// TwinCAT 3 PLC project OOP_PLC
// ProgramVersion: 3.1.4020.10
// libraries:
//   Tc2_Standard, * (Beckhoff Automation GmbH)
//   Tc2_System, * (Beckhoff Automation GmbH)
//   Tc3_Module, * (Beckhoff Automation GmbH)
//   VisuDialogs, * (System)
//   Tc3_System_DK,3.3.1.8,Beckhoff - DK
// project tree:
//   000 - General/ FB_RcvData.TcPOU, FB_RcvDataBuffer.TcPOU, GVL_MachineSettings.TcGVL, MAIN.TcPOU, P_System.TcPOU, visMain.TcVIS
//   010 - Machine Part 01/ FB_MachinePart01.TcPOU, ST_SettingMachinePart01.TcDUT, visSettingMachPart1.TcVIS
//   020 - Machine Part 02/ FB_MachinePart02.TcPOU, ST_SettingMachinePart02.TcDUT, visSettingMachPart2.TcVIS
//   100 - Network/ FB_CustomTcp.TcPOU, I_TcpClient.TcIO, I_TcpRcv.TcIO, SampleTcpClient.TcPOU, FB_SimpleTcpClient.TcPOU, SampleTcpServer.TcPOU, SampleUdpEchoServer.TcPOU, ST_Log.TcDUT, T_TcpRcv.TcDUT, U_IPAddr.TcDUT, U_Data.TcDUT
//   990 - NTO Standard/HResult/ F_Busy.TcPOU, F_Code.TcPOU, F_Fail.TcPOU, F_Success.TcPOU, GVL_HResultError.TcGVL, GVL_HResultSuccess.TcGVL
//   990 - NTO Standard/Object/ FB_Object.TcPOU, GVL_ObjectSetup.TcGVL, I_Object.TcIO, T_ErrorHistory.TcDUT
//   991 - NTO Actuators/010 - Cylinders/CylinderCollection/ FB_CylinderOneValveSpringRetX_2.TcPOU, FB_CylinderTwoValveRetX_3.TcPOU, txtCylinderTypes.TcTLO
//   991 - NTO Actuators/010 - Cylinders/ E_CylinderEnableMode.TcDUT, I_StandardCylinder.TcIO, ST_StandardCylinderSettings.TcDUT, txtLstCylinderEnableMode.TcTLO, visStandardCylinderSettings.TcVIS
//   991 - NTO Actuators/020 - Motors/MotorCollection/ FB_Motor.TcPOU, FB_MotorInverterFITYPE.TcPOU, txtMotorTypes.TcTLO
//   991 - NTO Actuators/020 - Motors/ E_MotorEnableMode.TcDUT, I_StandardMotor.TcIO, ST_StandardMotorSettings.TcDUT, txtLstMotorEnableMode.TcTLO, visStandardMotorSettings.TcVIS
//   / GlobalTextList.TcGTLO, PlcTask.TcTTO, Visualization Manager.TcVMO (not stored)
// real-time tasks:
//   TASK PlcTask: cycle T#1ms, priority 20, ADS port 350
//   TASK VISU_TASK: cycle T#200000us, priority 30, ADS port 351
// I/O:
//   DEVICE Device 1 (RT-Ethernet Adapter)

CONFIGURATION OOP_PLC
    RESOURCE PLC ON TwinCAT3
        TASK PlcTask(INTERVAL := T#1ms, PRIORITY := 20);
        PROGRAM MAIN WITH PlcTask : MAIN;
    END_RESOURCE
END_CONFIGURATION

// ---- 010 - Machine Part 01/ST_SettingMachinePart01.TcDUT
TYPE ST_SettingMachinePart01 :
STRUCT
    nMotorType : BYTE; //Motor type
    stMotorSettings : ST_StandardMotorSettings;
    nCylinderType : BYTE; //Cylinder type
    stCylinderSettings : ST_StandardCylinderSettings;
END_STRUCT
END_TYPE

// ---- 020 - Machine Part 02/ST_SettingMachinePart02.TcDUT
TYPE ST_SettingMachinePart02 :
STRUCT
    nCylinder1Type : BYTE; //Cylinder type
    stCylinder1Settings : ST_StandardCylinderSettings;
    nCylinder2Type : BYTE; //Cylinder type
    stCylinder2Settings : ST_StandardCylinderSettings;
END_STRUCT
END_TYPE

// ---- 100 - Network/ST_Log.TcDUT
TYPE ST_Log :
STRUCT
	nSocketID : UDINT;
	eTcpEvent : TCPIP_EVENT;
	sMessage : STRING;
END_STRUCT
END_TYPE

// ---- 100 - Network/T_TcpRcv.TcDUT
TYPE T_TcpRcv : POINTER TO FB_RcvDataBuffer; END_TYPE

// ---- 100 - Network/U_IPAddr.TcDUT
TYPE U_IPAddr :
UNION
	aIpAddr : ARRAY[0..3] OF BYTE;
	nIpAddr : UDINT;
END_UNION
END_TYPE

// ---- 100 - Network/U_Data.TcDUT
TYPE U_Data :
UNION
	sData : STRING(255);
	aData : ARRAY[0..255] OF BYTE;
END_UNION
END_TYPE

// ---- 990 - NTO Standard/Object/T_ErrorHistory.TcDUT
///Error history type
TYPE T_ErrorHistory : ARRAY[GVL_ObjectSetup.cErrorHistMin..GVL_ObjectSetup.cErrorHistMax] OF DWORD; END_TYPE

// ---- 991 - NTO Actuators/010 - Cylinders/E_CylinderEnableMode.TcDUT
{attribute 'qualified_only'}
{attribute 'strict'}
///Cylinder enable mode
TYPE E_CylinderEnableMode :
(
    eCylEnaOff,         ///Enable does not affect cylinder
	eCylEnaToHome,      ///When enable false, move cylinder to home
    eCylEnaToOut,       ///When enable false, move cylinder to out
    eCylEnaNoChanges    ///When enable false, cylinder keeps the position
);
END_TYPE

// ---- 991 - NTO Actuators/010 - Cylinders/ST_StandardCylinderSettings.TcDUT
///Standard cylinder settings
TYPE ST_StandardCylinderSettings :
STRUCT
    bSensorAtOut : BOOL; ///Cylinder has sensor at out
    tTimeToOrAtOut : TIME; ///Cylinder at or to out, bSensorOut = true: at out, bSensorOut = false: to out 
    bSensorAtHome : BOOL; ///Cylinder has sensor at home
    tTimeToOrAtHome : TIME; ///Cylinder at or to home, bSensorOut = true: at home, bSensorOut = false: to home
    eEnableMode : E_CylinderEnableMode; ///Cylinder enable mode
END_STRUCT
END_TYPE

// ---- 991 - NTO Actuators/020 - Motors/E_MotorEnableMode.TcDUT
{attribute 'qualified_only'}
{attribute 'strict'}
///Cylinder enable mode
TYPE E_MotorEnableMode :
(
    eMotorEnaOff,       ///Enable does not affect motor
    eMotorEnaAll,       ///When enable false, motor cannot move CW or CCW
    eMotorEnaAllowCW,   ///When enable false, motor can onlu move CW
    eMotorEnaAllowCCW   ///When enable false, motor can onlu move CCW   
);
END_TYPE

// ---- 991 - NTO Actuators/020 - Motors/ST_StandardMotorSettings.TcDUT
///Standard motor settings
TYPE ST_StandardMotorSettings :
STRUCT
    eEnableMode : E_MotorEnableMode; ///Enable mode
    nMaxSpeed : UINT; //Max speed in 0.1%
    nMaxAcc : UINT; //Max accelaration in FI dependent type
    nMaxDec : UINT; //Max deceleration in FI dependent type
END_STRUCT
END_TYPE

// ---- 000 - General/GVL_MachineSettings.TcGVL
{attribute 'qualified_only'}
VAR_GLOBAL PERSISTENT
    stSettingsMach01_1 : ST_SettingMachinePart01 := (nMotorType := 0, nCylinderType := 1);
    stSettingsMach01_2 : ST_SettingMachinePart01 := (nMotorType := 1, nCylinderType := 0);
    stSettingsMach02_1 : ST_SettingMachinePart02 := (
		nCylinder1Type := 0, stCylinder1Settings := (bSensorAtOut := TRUE, eEnableMode := E_CylinderEnableMode.eCylEnaToHome),
		nCylinder2Type := 1, stCylinder2Settings := (bSensorAtOut := FALSE, eEnableMode := E_CylinderEnableMode.eCylEnaToOut));
    stSettingsMach02_2 : ST_SettingMachinePart02 := (nCylinder1Type := 1, nCylinder2Type := 0);
END_VAR

// ---- 990 - NTO Standard/HResult/GVL_HResultError.TcGVL
{attribute 'qualified_only'}
VAR_GLOBAL CONSTANT
    cHR_ErrGeneral : HRESULT := UDINT_TO_DINT(16#A0000000); //Fail with general error
    cHR_ErrInvalidParameter : HRESULT := UDINT_TO_DINT(16#A0000001); //Fail with invalid parameters    
	cHR_ErrConnect : HRESULT := UDINT_TO_DINT(16#A0000002); //Fail, when trying to connect
	cHR_ErrAllocSocket : HRESULT := UDINT_TO_DINT(16#A0000003); //Fail, when allocating a socket
	cHR_ErrNotConnected : HRESULT := UDINT_TO_DINT(16#A0000002); //Fail, not connected
END_VAR

// ---- 990 - NTO Standard/HResult/GVL_HResultSuccess.TcGVL
{attribute 'qualified_only'}
VAR_GLOBAL CONSTANT
    cHR_SuccesDone : HRESULT := 16#20000001; //Successfully done
    cHR_SuccesBusy : HRESULT := 16#20000002; //Busy, keep calling to wait for done or error    
END_VAR

// ---- 990 - NTO Standard/Object/GVL_ObjectSetup.TcGVL
{attribute 'qualified_only'}
VAR_GLOBAL CONSTANT
    cErrorHistMin : INT := 0; ///Error history array bound minimum
    cErrorHistMax : INT := 10; ///Error history array bound maximum
END_VAR

// ---- 100 - Network/I_TcpClient.TcIO
{attribute 'c++_compatible'}
INTERFACE I_TcpClient EXTENDS I_Object

METHOD PUBLIC Connect : HRESULT
VAR_INPUT
	uIPAddr : U_IPAddr;
	nPort : UINT;
	{warning 'Implemented with POINTER TO, until Beckhoff comes with solution to why Interface call crashes app'}
	ipRcvData : T_TcpRcv;//I_TcpRcv; 
END_VAR
END_METHOD

PROPERTY DataLogging : BOOL
GET
END_GET
SET
END_SET
END_PROPERTY

METHOD PUBLIC Disconnect : HRESULT
VAR_INPUT
END_VAR
END_METHOD

PROPERTY EventLogging : BOOL
GET
END_GET
SET
END_SET
END_PROPERTY

PROPERTY IpAddress : U_IPAddr
GET
END_GET
END_PROPERTY

PROPERTY IsConnected : BOOL
GET
END_GET
END_PROPERTY

PROPERTY Port : UINT
GET
END_GET
END_PROPERTY

METHOD SendData : HRESULT
VAR_INPUT
	nData : UDINT;
	pData : PVOID;
END_VAR
END_METHOD

PROPERTY SendingData : BOOL
GET
END_GET
END_PROPERTY

END_INTERFACE

// ---- 100 - Network/I_TcpRcv.TcIO
{attribute 'c++_compatible'}
INTERFACE I_TcpRcv

METHOD NewData : HRESULT
VAR_INPUT
	nData	: UDINT;
	pData	: PVOID;
END_VAR
END_METHOD

END_INTERFACE

// ---- 990 - NTO Standard/Object/I_Object.TcIO
{attribute 'c++_compatible'}
///Base object interface
INTERFACE I_Object

//Cycle Task, do not override this methode cyclic code is placed in M_Control
METHOD CycleTask
VAR_INPUT
END_VAR
END_METHOD

///Error, do not implement property override
PROPERTY Error : BOOL
GET
END_GET
END_PROPERTY

///Error id, do not implement property override
PROPERTY ErrorID : DWORD
GET
END_GET
END_PROPERTY

///Pointer to error history, do not implement property override
PROPERTY Errors : POINTER TO T_ErrorHistory
GET
END_GET
END_PROPERTY

///Name, do not implement property override
PROPERTY PUBLIC Name : String(50)
GET
END_GET
END_PROPERTY

///Reset error, allways call super
METHOD Reset
VAR_INPUT
END_VAR
END_METHOD

///Version,do not implement property override
PROPERTY PUBLIC Version : String(8)
GET
END_GET
END_PROPERTY

END_INTERFACE

// ---- 991 - NTO Actuators/010 - Cylinders/I_StandardCylinder.TcIO
{attribute 'c++_compatible'}
///Standard cylinder
INTERFACE I_StandardCylinder EXTENDS I_Object

///Cylinder at home position
PROPERTY AtHome : BOOL
GET
END_GET
END_PROPERTY

///Cylinder at out position
PROPERTY AtOut : BOOL
GET
END_GET
END_PROPERTY

///Enable cylinder to change position
PROPERTY Enable : BOOL
GET
END_GET
SET
END_SET
END_PROPERTY

METHOD MoveHome
VAR_INPUT
END_VAR
END_METHOD

METHOD MoveOut
VAR_INPUT
END_VAR
END_METHOD

///Pointer to settings, should be set at FB_init but can be modified with set accessor if needed
PROPERTY Settings : POINTER TO ST_StandardCylinderSettings
GET
END_GET
SET
END_SET
END_PROPERTY

END_INTERFACE

// ---- 991 - NTO Actuators/020 - Motors/I_StandardMotor.TcIO
{attribute 'c++_compatible'}
///Standard motor
INTERFACE I_StandardMotor EXTENDS I_Object

///Accelaration in FI dependent type
PROPERTY Acc : UINT
GET
END_GET
SET
END_SET
END_PROPERTY

///Move motor CCW
PROPERTY CCW : BOOL
GET
END_GET
SET
END_SET
END_PROPERTY

///Move motor CW
PROPERTY CW : BOOL
GET
END_GET
SET
END_SET
END_PROPERTY

///Deceleration in FI dependent type
PROPERTY Dec : UINT
GET
END_GET
SET
END_SET
END_PROPERTY

///Enable Motor
PROPERTY Enable : BOOL
GET
END_GET
SET
END_SET
END_PROPERTY

///Limit counter-clockwise rotation
PROPERTY LimitCCW : BOOL
GET
END_GET
SET
END_SET
END_PROPERTY

///Limit clockwise rotation
PROPERTY LimitCW : BOOL
GET
END_GET
SET
END_SET
END_PROPERTY

///Pointer to settings, should be set at FB_init but can be modified with set accessor if needed
PROPERTY Settings : POINTER TO ST_StandardMotorSettings
GET
END_GET
SET
END_SET
END_PROPERTY

///Motor speed in 0.1 % 
PROPERTY Speed : UINT
GET
END_GET
SET
END_SET
END_PROPERTY

END_INTERFACE

// ---- 000 - General/MAIN.TcPOU
PROGRAM MAIN
//Beckhoff.dk, System_DK 
VAR
	bReset: BOOL;
	bWrite: BOOL;
END_VAR
VAR
	fbTcpClient : FB_SimpleTcpClient;
	bLogON : BOOL;
	bConnect : BOOL;
	bDisconnect : BOOL;
	bSendData :BOOL;	
	nResConnect : HRESULT;
	nResDisconnect : HRESULT;
	nResSendData : HRESULT;
	bIsConnected : BOOL;
	bSendingData : BOOL;
	uIP : U_IPAddr := (aIpAddr := [14,1,168,192]);
	sData : U_Data;
	nCnt : UDINT;
	
END_VAR

VAR
	fbRcvData2 : FB_RcvData;
	fbRcvData : FB_RcvDataBuffer(ipSubscriber := ADR(fbRcvData2));
END_VAR

(*
VAR CONSTANT
    cMaxObjects1 : INT := 3;
END_VAR
VAR
    fbMach01_1 : FB_MachinePart01(pSettings := ADR(GVL_MachineSettings.stSettingsMach01_1));   
    fbMach01_2 : FB_MachinePart01(pSettings := ADR(GVL_MachineSettings.stSettingsMach01_2));
    fbMach02_1 : FB_MachinePart02(pSettings := ADR(GVL_MachineSettings.stSettingsMach02_1));
    fbMach02_2 : FB_MachinePart02(pSettings := ADR(GVL_MachineSettings.stSettingsMach02_2));
END_VAR
VAR
    nLoop : INT;
    aObjects : ARRAY[0..cMaxObjects1] OF I_Object := [fbMach01_1,fbMach01_2,fbMach02_1,fbMach02_2];
END_VAR
*)

//Beckhoff.dk standard system
P_System(bWritePersistent:= bWrite, bReset:= bReset); 

fbTcpClient.CycleTask();
fbTcpClient.DataLogging := bLogON;

IF bConnect THEN
	nResConnect := fbTcpClient.Connect(uIPAddr := uIP, nPort := 9990, ipRcvData :=  ADR(fbRcvData));
	bConnect := FALSE;
END_IF

IF bDisconnect THEN
	nResDisconnect := fbTcpClient.Disconnect();
	bDisconnect := FALSE;
END_IF

bIsConnected := fbTcpClient.IsConnected;
bSendingData := fbTcpClient.SendingData;


IF bIsConnected AND bSendData AND NOT(bSendingData) THEN
	sData.sData := Tc2_Standard.CONCAT('Cnt: ', Tc2_Standard.CONCAT(UDINT_TO_STRING(nCnt),'$n$r'));
	nCnt := nCnt + 1;
	fbTcpClient.SendData(pData := ADR(sData), nData := INT_TO_UDINT(Tc2_Standard.LEN(sData.sData)));
	sData.sData := Tc2_Standard.CONCAT('Cnt: ', Tc2_Standard.CONCAT(UDINT_TO_STRING(nCnt),'$n$r'));
	nCnt := nCnt + 1;
	fbTcpClient.SendData(pData := ADR(sData), nData := INT_TO_UDINT(Tc2_Standard.LEN(sData.sData)));
END_IF



(*
FOR nLoop := 0 TO cMaxObjects1 DO
    IF aObjects[nLoop] <> 0 THEN
        aObjects[nLoop].CycleTask();
	END_IF
END_FOR
*)

END_PROGRAM

// ---- 100 - Network/FB_SimpleTcpClient.TcPOU
{attribute 'c++_compatible'}
FUNCTION_BLOCK FB_SimpleTcpClient EXTENDS FB_Object IMPLEMENTS ITcIoTcpProtocolRecv, I_TcpClient
VAR
	{attribute 'TcInitSymbol'}
	oid : OTCID;
	{attribute 'hide'}
	ipTcp : ITcIoTcpProtocol;
	{attribute 'hide'}
	nSocketID : UDINT;
	{attribute 'hide'}	
	nPort : UINT;
	{attribute 'hide'}
	uIP : U_IPAddr;
	{attribute 'hide'}
	fbDelayBeforeConnected : Tc2_Standard.TON;
	{attribute 'hide'}
	bSendData : BOOL;
	
END_VAR
///Log
VAR
	aEventsLog : ARRAY[0..cMaxEventsLogEntries] OF ST_Log;
	nEventsLogEntries : UINT := 0;
	aRcvDataLog : ARRAY[0..cMaxDataLogEntries] OF STRING(cMaxDataLogEntryLength);
	nRcvDataEntries : UINT;
	{attribute 'hide'}
	bEventLog : BOOL := TRUE;	
	{attribute 'hide'}
	bDataLog : BOOL := FALSE;	
	{warning 'Implemented with POINTER TO, until Beckhoff comes with solution to why Interface call crashes app'}
	{attribute 'hide'}
	ipReciever : T_TcpRcv;//I_TcpRcv;
END_VAR
VAR CONSTANT
	cMaxEventsLogEntries : UINT := 100;
	cMaxDataLogEntries : UDINT := 25;
	cMaxDataLogEntryLength : UDINT := 255;
END_VAR

METHOD PUBLIC Connect : HRESULT
VAR_INPUT
	uIPAddr : U_IPAddr;
	nPort : UINT;
	ipRcvData : T_TcpRcv;//I_TcpRcv;
END_VAR
IF nSocketID <> 0 OR ipTcp = 0 THEN
	Connect := GVL_HResultError.cHR_ErrGeneral;
	RETURN;
END_IF

IF uIPAddr.nIpAddr = 0 OR nPort = 0 THEN
	Connect := GVL_HResultError.cHR_ErrInvalidParameter;
	RETURN;
END_IF
bSendData := 0;

//Open socket
IF Tc3_Module.SUCCEEDED(ipTcp.AllocSocket(ipRecv := THIS^, socketId := nSocketID)) THEN
	
	IF Tc3_Module.FAILED(ipTcp.Connect(socketId := nSocketID, ipRemoteAddress := uIPAddr.nIpAddr, tcpPort := nPort)) THEN
		ipTcp.FreeSocket(nSocketID);
		nSocketID := 0;
		Connect := GVL_HResultError.cHR_ErrConnect;
		fbDelayBeforeConnected.IN := FALSE;
	ELSE
		Connect := GVL_HResultSuccess.cHR_SuccesDone;
		fbDelayBeforeConnected.IN := TRUE;
		uIP := uIPAddr;
		nPort := nPort;
		ipReciever := ipRcvData;
	END_IF 
	
ELSE
	
	nSocketID := 0;
	Connect := GVL_HResultError.cHR_ErrAllocSocket;
	fbDelayBeforeConnected.IN := FALSE;
	
END_IF
END_METHOD

METHOD INTERNAL Control
IF ipTcp <> 0 THEN
	ipTcp.CheckReceived();
	fbDelayBeforeConnected();
	fbDelayBeforeConnected.PT := T#10000MS;
END_IF;
END_METHOD

PROPERTY DataLogging : BOOL
GET
DataLogging := bDataLog;
END_GET
SET
bDataLog := DataLogging;
END_SET
END_PROPERTY

METHOD PUBLIC Disconnect : HRESULT
VAR_INPUT
END_VAR
IF nSocketID = 0 OR ipTcp = 0 THEN
	Disconnect := GVL_HResultError.cHR_ErrGeneral;
	RETURN;
END_IF

//Close socket
IF Tc3_Module.SUCCEEDED(ipTcp.IsConnected(nSocketID)) THEN
	ipTcp.Close(nSocketID);
	ipTcp.CheckReceived();
END_IF
fbDelayBeforeConnected.IN := FALSE;
ipTcp.FreeSocket(nSocketID);
nSocketID := 0;

uIP.nIpAddr := 0;
nPort := 0;
bSendData := 0;
ipReciever := 0;

Disconnect := GVL_HResultSuccess.cHR_SuccesDone;
END_METHOD

PROPERTY EventLogging : BOOL
GET
EventLogging := bEventLog;
END_GET
SET
bEventLog := EventLogging;
END_SET
END_PROPERTY

METHOD FB_exit : BOOL
VAR_INPUT
	bInCopyCode : BOOL; // if TRUE, the exit method is called for exiting an instance that is copied afterwards (online change).
END_VAR
IF ipTcp <> 0 THEN
	IF nSocketID <> 0 THEN
		IF Tc3_Module.SUCCEEDED(ipTcp.IsConnected(nSocketID)) THEN
			ipTcp.Close(nSocketID);
			ipTcp.CheckReceived();
		END_IF
		ipTcp.FreeSocket(nSocketID);
		nSocketID := 0;
	ELSE
		FB_exit := TRUE;
	END_IF
ELSE
	FB_exit := FALSE;	
END_IF
END_METHOD

METHOD FB_init : BOOL
VAR_INPUT
	bInitRetains : BOOL; // if TRUE, the retain variables are initialized (warm start / cold start)
	bInCopyCode : BOOL;  // if TRUE, the instance afterwards gets moved into the copy code (online change)
END_VAR
VAR
	ipSrv : ITComObjectServer;
END_VAR
sName := 'FB_SimpleTcpClient';
sVersion := '1.0.0.0';

IF Tc3_Module.FW_ObjMgr_GetObjectServer(oidApp := _AppInfo.ObjId, pipSrv := ADR(ipSrv)) = Tc3_Module.S_OK THEN
	
	IF ipSrv.TcQueryObjectInterface(oid := oid, iid := IID_ITcIoTcpProtocol, ADR(ipTcp)) = Tc3_Module.S_OK THEN
		FB_init := TRUE;
	ELSE
		FB_init := FALSE;
	END_IF
	ipSrv.TcRelease();
	ipSrv := 0;
ELSE
	FB_init := FALSE;
END_IF
END_METHOD

PROPERTY IpAddress : U_IPAddr
GET
IpAddress := uIP;
END_GET
END_PROPERTY

PROPERTY IsConnected : BOOL
GET
IF nSocketID <> 0 AND ipTcp <> 0 AND fbDelayBeforeConnected.Q THEN
	IsConnected := Tc3_Module.SUCCEEDED(ipTcp.IsConnected(nSocketID));
ELSE
	IsConnected := FALSE;
END_IF
END_GET
END_PROPERTY

PROPERTY Port : UINT
GET
Port := nPort;
END_GET
END_PROPERTY

{attribute 'c++_compatible'}
{attribute 'signature_flag' := '33554688'}
{attribute 'pack_mode' := '4'}
{attribute 'show'}
{attribute 'minimal_input_size' := '4'}
{attribute 'checksuperglobal'}
METHOD ReceiveData : HRESULT
VAR_INPUT
	socketId	: UDINT;
	nData	: UDINT;
	pData	: PVOID;
END_VAR
VAR
	nRes : HRESULT;
END_VAR
ReceiveData := Tc3_Module.S_OK;
//Log data, if enabled
IF bDataLog THEN
	
	Tc2_System.MEMCPY(ADR(aRcvDataLog[nRcvDataEntries]),pData,MIN(cMaxDataLogEntryLength,nData));
	nRcvDataEntries := nRcvDataEntries + 1;
	
	IF nRcvDataEntries > cMaxDataLogEntries THEN
		nRcvDataEntries := 0;
	END_IF
	
END_IF

//Notify listeners
IF ipReciever <> 0 THEN 
	{warning 'Implemented with POINTER TO, until Beckhoff comes with solution to why Interface call crashes app'}
	ipReciever^.NewData(nData := nData, pData := pData);
END_IF
END_METHOD

{attribute 'c++_compatible'}
{attribute 'signature_flag' := '33554688'}
{attribute 'pack_mode' := '4'}
{attribute 'show'}
{attribute 'minimal_input_size' := '4'}
{attribute 'checksuperglobal'}
METHOD ReceiveEvent : HRESULT
VAR_INPUT
	socketId	: UDINT;
	tcpEvent	: TCPIP_EVENT;
END_VAR
ReceiveEvent := Tc3_Module.S_OK;
IF bEventLog THEN
	aEventsLog[nEventsLogEntries].eTcpEvent := tcpEvent;
	aEventsLog[nEventsLogEntries].nSocketID := socketId;
	nEventsLogEntries := nEventsLogEntries + 1;
	IF nEventsLogEntries > cMaxEventsLogEntries THEN
		nEventsLogEntries := 0;
	END_IF
END_IF

CASE tcpEvent OF
	TCPIP_EVENT.TCPIP_EVENT_CONN_CLOSED :
		THIS^.Disconnect();
	TCPIP_EVENT.TCPIP_EVENT_RESET :
		THIS^.Disconnect();
	TCPIP_EVENT.TCPIP_EVENT_DATA_SENT :
		bSendData := FALSE;
	TCPIP_EVENT.TCPIP_EVENT_CONN_ESTABLISHED :
		fbDelayBeforeConnected.PT := T#0MS;
END_CASE
END_METHOD

METHOD SendData : HRESULT
VAR_INPUT
	nData : UDINT;
	pData : PVOID;
END_VAR
VAR
	nSendData : UDINT;
END_VAR
IF uIP.nIpAddr = 0 OR nPort = 0 THEN
	SendData := GVL_HResultError.cHR_ErrInvalidParameter;
	RETURN;
END_IF

IF NOT(THIS^.IsConnected) THEN
	SendData := GVL_HResultError.cHR_ErrNotConnected;
	RETURN;
END_IF

SendData := ipTcp.SendData(socketId := nSocketID, nData := nData, pData := pData, nSendData := nSendData);
bSendData := 1;
END_METHOD

PROPERTY SendingData : BOOL
GET
SendingData := bSendData;
END_GET
END_PROPERTY

{attribute 'c++_compatible'}
{attribute 'signature_flag' := '33554688'}
{attribute 'pack_mode' := '4'}
{attribute 'show'}
{attribute 'minimal_input_size' := '4'}
{attribute 'checksuperglobal'}
METHOD TcAddRef : UDINT
END_METHOD

{attribute 'c++_compatible'}
{attribute 'signature_flag' := '33554688'}
{attribute 'pack_mode' := '4'}
{attribute 'show'}
{attribute 'minimal_input_size' := '4'}
{attribute 'checksuperglobal'}
METHOD TcQueryInterface : HRESULT
VAR_INPUT
	iid	: REFERENCE TO IID;
	pipItf	: POINTER TO PVOID;
END_VAR
END_METHOD

{attribute 'c++_compatible'}
{attribute 'signature_flag' := '33554688'}
{attribute 'pack_mode' := '4'}
{attribute 'show'}
{attribute 'minimal_input_size' := '4'}
{attribute 'checksuperglobal'}
METHOD TcRelease : UDINT
END_METHOD

END_FUNCTION_BLOCK

// ---- 990 - NTO Standard/Object/FB_Object.TcPOU
{attribute 'c++_compatible'}
///Object base FB for all FB's
FUNCTION_BLOCK FB_Object IMPLEMENTS I_Object
VAR
    sName : STRING(50) := 'FB_Object'; //FB Name
    sVersion : STRING(8) := '1.0.0.0'; //FB Version
    bFirstPass : BOOL := FALSE; //First pass done
    bError : BOOL := FALSE; //Error
    nErrorID : DWORD := 0; //Error id
    aErrors : T_ErrorHistory; //Error history
END_VAR

///Add error to error history
METHOD PROTECTED AddError
VAR_INPUT
	nErrorID : DWORD; //Error ID
END_VAR
VAR
	nAddErrorLoop : INT;
END_VAR
FOR nAddErrorLoop := GVL_ObjectSetup.cErrorHistMax TO (GVL_ObjectSetup.cErrorHistMin + 1) BY -1 DO
	aErrors[nAddErrorLoop] := aErrors[nAddErrorLoop - 1];
END_FOR
aErrors[GVL_ObjectSetup.cErrorHistMin] := nErrorID;
END_METHOD

///Control, override to get cyclic task in FB
METHOD INTERNAL Control
VAR_INPUT
END_VAR
END_METHOD

//Cycle Task, do not override this methode cyclic code is placed in M_Control 
METHOD CycleTask
IF NOT(bFirstPass) THEN
    bFirstPass := Init() = GVL_HResultSuccess.cHR_SuccesDone;
    IF NOT(bFirstPass) THEN
        RETURN;
	END_IF
END_IF
Control();
END_METHOD

(*Error, do not implement property override*)
PROPERTY Error : BOOL
GET
Error := bError;
END_GET
END_PROPERTY

(*error id, do not implement property override*)
PROPERTY ErrorID : DWORD
GET
ErrorID := nErrorID;
END_GET
END_PROPERTY

(*Pointer to error history, do not implement property override*)
PROPERTY Errors : POINTER TO T_ErrorHistory
GET
Errors := ADR(aErrors);
END_GET
END_PROPERTY

METHOD FB_init : BOOL
VAR_INPUT
	bInitRetains : BOOL; // if TRUE, the retain variables are initialized (warm start / cold start)
	bInCopyCode : BOOL;  // if TRUE, the instance afterwards gets moved into the copy code (online change)
END_VAR
bFirstPass := FALSE;
END_METHOD

///Initialize FB, Override to do custom initialize, no need to call super
METHOD INTERNAL Init : HRESULT
Init := GVL_HResultSuccess.cHR_SuccesDone;
END_METHOD

(*Name, do not implement property override*)
PROPERTY Name : STRING(50)
GET
Name := sName;
END_GET
END_PROPERTY

(*Reset error, allways call super*)
METHOD Reset
bError := FALSE;
nErrorID := 0;
END_METHOD

///Set error on the Object and add entry to error history
METHOD PROTECTED SetError
VAR_INPUT
	nErrorID : DWORD; //Error ID
END_VAR
VAR
    nSetErrorLoop : INT;
END_VAR
IF NOT(bError) THEN
	bError := TRUE;
	THIS^.nErrorID := nErrorID;
	FOR nSetErrorLoop := GVL_ObjectSetup.cErrorHistMax TO (GVL_ObjectSetup.cErrorHistMin + 1) BY -1 DO
    	aErrors[nSetErrorLoop] := aErrors[nSetErrorLoop - 1];
	END_FOR
	aErrors[GVL_ObjectSetup.cErrorHistMin] := nErrorID;
END_IF
END_METHOD

(*Version,do not implement property override*)
PROPERTY Version : STRING(8)
GET
Version := sVersion;
END_GET
END_PROPERTY

END_FUNCTION_BLOCK

// ---- 000 - General/FB_RcvData.TcPOU
{attribute 'c++_compatible'}
FUNCTION_BLOCK FB_RcvData IMPLEMENTS I_TcpRcv
VAR
	nRcvCnt : UDINT;
	sData : STRING(255);
END_VAR

METHOD NewData : HRESULT
VAR_INPUT
	nData	: UDINT;
	pData	: PVOID;
END_VAR
IF nData <> 0 AND pData <> 0 THEN
	nRcvCnt := nRcvCnt + 1;
	Tc2_System.MEMCPY(destAddr := ADR(sData),srcAddr := pData, n := MIN(255,nData));
END_IF
END_METHOD

END_FUNCTION_BLOCK

// ---- 000 - General/FB_RcvDataBuffer.TcPOU
{attribute 'c++_compatible'}
FUNCTION_BLOCK FB_RcvDataBuffer IMPLEMENTS I_TcpRcv
VAR
	nRcvCnt : UDINT;
	sNewData : STRING(1000);
	nNewDataCnt : UDINT;
	
	nBufferPos : UDINT := 0;
	nState : USINT;
	
	aRcvDataBuffer : ARRAY[0..cMaxData] OF BYTE;
	aDataBuffer : ARRAY[0..cMaxData] OF BYTE;
	
	ipSubscriber : T_TcpRcv;
	
END_VAR
VAR CONSTANT
	cMaxData : UDINT := 1000;
END_VAR

METHOD FB_init : BOOL
VAR_INPUT
	bInitRetains : BOOL; // if TRUE, the retain variables are initialized (warm start / cold start)
	bInCopyCode : BOOL;  // if TRUE, the instance afterwards gets moved into the copy code (online change)
	ipSubscriber : T_TcpRcv;
END_VAR
THIS^.ipSubscriber := ipSubscriber;
END_METHOD

METHOD NewData : HRESULT
VAR_INPUT
	nData	: UDINT;
	pData	: PVOID;
END_VAR
VAR
	bExit : BOOL;
	nDataLength : UDINT;
	nLoopNewData : UDINT;
	nPosStart : UDINT;
END_VAR
IF nData = 0 OR pData = 0 THEN
	NewData := GVL_HResultError.cHR_ErrInvalidParameter;
	RETURN;
END_IF

nRcvCnt := nRcvCnt + 1;
nDataLength := MIN(nData, cMaxData);

Tc2_System.MEMSET(destAddr := ADR(aRcvDataBuffer), fillByte := 0, n := SIZEOF(aRcvDataBuffer));
Tc2_System.MEMCPY(destAddr := ADR(aRcvDataBuffer), srcAddr := pData, n := nDataLength); 

bExit := FALSE;
nPosStart := 0; 

REPEAT
	
	CASE nState OF 
		0 : //Waiting for STX	
			FOR nLoopNewData := 0 TO nDataLength - 1 DO
				IF aRcvDataBuffer[nLoopNewData] = 16#02 THEN
					nPosStart := nLoopNewData;
					nState := 1;
					nBufferPos := 0;
					EXIT;
				END_IF
			END_FOR
			IF nState = 0 THEN
				bExit := TRUE;
			END_IF
			
		1 : //Check for ETX
			FOR nLoopNewData := nPosStart TO nDataLength - 1 DO		
		
				aDataBuffer[nBufferPos] := aRcvDataBuffer[nLoopNewData];
				nBufferPos := nBufferPos + 1;
				
				IF aRcvDataBuffer[nLoopNewData] = 16#03 THEN
					nState := 2;
					EXIT;
				END_IF
				
			END_FOR
			
			IF nState = 1 THEN
				bExit := TRUE;
			END_IF
			
		2 : //Copy telegram to buffer and then full to newdata rcv
			FOR nLoopNewData := 0 TO nBufferPos DO
				sNewData[nLoopNewData] := aDataBuffer[nLoopNewData];
			END_FOR
			
			sNewData[nBufferPos] := 0;
			
			IF ipSubscriber <> 0 THEN
				ipSubscriber^.NewData(pData := ADR(sNewData), nData := nBufferPos);
			END_IF
			
			nNewDataCnt := nNewDataCnt + 1;
			
			nBufferPos := 0;
			nState := 0;
			bExit := TRUE;
			
		ELSE
			
			nState := 0;
			bExit := TRUE;
		
	END_CASE
	
UNTIL
	bExit
END_REPEAT
END_METHOD

END_FUNCTION_BLOCK

// ---- 000 - General/P_System.TcPOU
PROGRAM P_System
VAR_INPUT
	bWritePersistent: BOOL;
	bReset: BOOL;
END_VAR
VAR_OUTPUT
	bEtherCAT_Ok: BOOL;
	bError: BOOL;
	nErrorID: UDINT;
END_VAR
VAR
	nAlive: UDINT;
	bFirstScan: BOOL:= TRUE;

//******************************************************************************
// System	
//******************************************************************************
	fbSystemDK: Tc3_System_DK.FB_SystemDK;
	ipSystemDK: Tc3_System_DK.I_SystemDK:= fbSystemDK;
	stSystemDK: Tc3_System_DK.ST_SystemDK;  
	
//******************************************************************************
// EtherCAT
//******************************************************************************
	fbEtherCATStatusDK: Tc3_System_DK.FB_EtherCATStatusDK;
	ipEtherCATStatusDK: Tc3_System_DK.I_EtherCATStatusDK:= fbEtherCATStatusDK;
	stEtherCATStatusDK: Tc3_System_DK.ST_EtherCATStatusDK;
	
//******************************************************************************
// Persistent
//******************************************************************************
	fbWritePersistentDataDK: Tc3_System_DK.FB_WritePersistentDataDK;
	ipWritePersistentDataDK: Tc3_System_DK.I_WritePersistentDataDK:= fbWritePersistentDataDK;
	stWritePersistentDataDK: Tc3_System_DK.ST_WritePersistentDataDK;
	
//******************************************************************************
// NovRam
//******************************************************************************
	fbNovRamDK: Tc3_System_DK.FB_NovRamDK;
	ipNovRamDK: Tc3_System_DK.I_NovRamDK:= fbNovRamDK;
	stNovRam: Tc3_System_DK.ST_NovRamDK;	
	
END_VAR

nAlive:= nAlive +1;

// Call actions
IF bFirstScan THEN
	A_Init();
ELSE
	A_Error();
	A_Prg();
END_IF

ACTION A_Error:
//******************************************************************************
// Error handling
//******************************************************************************
bError:= FALSE;
IF ipSystemDK.P_bError THEN
	bError:= TRUE;
END_IF
IF ipEtherCATStatusDK.P_bError THEN
	bError:= TRUE;
END_IF
IF ipWritePersistentDataDK.P_bError THEN
	bError:= TRUE;
END_IF
IF ipNovRamDK.P_bError THEN
	bError:= TRUE;
END_IF

nErrorID:= 16#0000;
IF ipSystemDK.P_bError THEN
	nErrorID:= ipSystemDK.P_nErrorID;
END_IF
IF ipEtherCATStatusDK.P_bError THEN
	nErrorID:= ipEtherCATStatusDK.P_nErrorID;
END_IF
IF ipWritePersistentDataDK.P_bError THEN
	nErrorID:= ipWritePersistentDataDK.P_nErrorID;
END_IF
IF ipNovRamDK.P_bError THEN
	nErrorID:= ipNovRamDK.P_nErrorID;
END_IF
END_ACTION

ACTION A_Init:


bFirstScan:= FALSE;
END_ACTION

ACTION A_Prg:
//	The result of the method is an unsigned double integer
//	0 = idle 
//	1 = coupled
//	2 = starting
//	3 = running
//	4 = aborted
// 	5 = no hardware connected
//  6 = Spare
//	7 = pointer or index error
//	8 = mapping error
//	9 = parameter error
//	10 = complete
//	Any other number = ErrorID


//******************************************************************************
// System
//******************************************************************************

// Call methods
stSystemDK.arr_nStatus[1]:= ipSystemDK.M_nEnable();
stSystemDK.arr_nStatus[2]:= ipSystemDK.M_nCerHost(bEnable:= stSystemDK.bCerHost_Enable, bDisable:= stSystemDK.bCerHost_Disable);
stSystemDK.arr_nStatus[3]:= ipSystemDK.M_nReset(bExecute:= bReset);

// Get property
stSystemDK.bReady:= ipSystemDK.P_bReady;
stSystemDK.bError:= ipSystemDK.P_bError;
stSystemDK.nErrorID:= ipSystemDK.P_nErrorID;
stSystemDK.bIs_CE_Device:= ipSystemDK.P_bIs_CE_Device;
stSystemDK.nAdsPort:= ipSystemDK.P_nAdsPort;
stSystemDK.nCycleTime:= ipSystemDK.P_nCycleTime;
stSystemDK.bIs_ARM:= ipSystemDK.P_bIs_ARM;
stSystemDK.bIs_x86:= ipSystemDK.P_bIs_x86;
stSystemDK.bIs_x64:= ipSystemDK.P_bIs_x64;
stSystemDK.sTwinCAT_Version:= ipSystemDK.P_sTwinCAT_Version;
stSystemDK.stDeviceIdentificationEx:= ipSystemDK.P_stDeviceIdentificationEx;

//******************************************************************************
// EtherCAT
//******************************************************************************

// Call methods
stEtherCATStatusDK.arr_nStatus[1]:= ipEtherCATStatusDK.M_nEnable(bExecute:= TRUE);
stEtherCATStatusDK.arr_nStatus[2]:= ipEtherCATStatusDK.M_nReset(bExecute:= bReset);

// Get property
stEtherCATStatusDK.bReady:= ipEtherCATStatusDK.P_bReady;
stEtherCATStatusDK.bError:= ipEtherCATStatusDK.P_bError;
stEtherCATStatusDK.nErrorID:= ipEtherCATStatusDK.P_nErrorID;
stEtherCATStatusDK.bWireBroke:= ipEtherCATStatusDK.P_bWireBroke;
stEtherCATStatusDK.nDevState:= ipEtherCATStatusDK.P_nDevState;
stEtherCATStatusDK.nSlaveCount:= ipEtherCATStatusDK.P_nSlaveCount;
stEtherCATStatusDK.nCfgSlaveCount:= ipEtherCATStatusDK.P_nCfgSlaveCount;

// EtherCAT status
bEtherCAT_Ok:= ipEtherCATStatusDK.P_bReady;

//******************************************************************************
// Persistent
//******************************************************************************

// Set proporty
ipWritePersistentDataDK.P_eSUPS_Mode:= Tc3_System_DK.eSUPS_WrPersistData_Shutdown;

// Call methods
stWritePersistentDataDK.arr_nStatus[1]:= ipWritePersistentDataDK.M_nEnable(bExecute:= TRUE, tLogTimePuls:= T#10M);
stWritePersistentDataDK.arr_nStatus[2]:= ipWritePersistentDataDK.M_nWrite(bExecute:= bWritePersistent);
stWritePersistentDataDK.arr_nStatus[3]:= ipWritePersistentDataDK.M_n1_second_UPS(bExecute:= TRUE);
stWritePersistentDataDK.arr_nStatus[4]:= ipWritePersistentDataDK.M_nReset(bExecute:= bReset);

// Get property
stWritePersistentDataDK.bReady:= ipWritePersistentDataDK.P_bReady;
stWritePersistentDataDK.bError:= ipWritePersistentDataDK.P_bError;
stWritePersistentDataDK.nErrorID:= ipWritePersistentDataDK.P_nErrorID;
stWritePersistentDataDK.bBusy:= ipWritePersistentDataDK.P_bBusy;
stWritePersistentDataDK.nWriteCNT:= ipWritePersistentDataDK.P_nWriteCNT;

(*

//******************************************************************************
// NovRam
//******************************************************************************

// Call methods
stNovRam.arr_nStatus[1]:= ipNovRamDK.M_nEnable(bExecute:= TRUE, nDevId:= 2, nMB_Offset:= 0, nMB_Size:= 2048);
stNovRam.arr_nStatus[2]:= ipNovRamDK.M_nReset(bExecute:= bReset);

// Get property
stNovRam.bReady:= ipNovRamDK.P_bReady;
stNovRam.bError:= ipNovRamDK.P_bError;
stNovRam.nErrorID:= ipNovRamDK.P_nErrorID;

*)
END_ACTION

END_PROGRAM

// ---- 010 - Machine Part 01/FB_MachinePart01.TcPOU
{attribute 'c++_compatible'}
FUNCTION_BLOCK FB_MachinePart01 EXTENDS FB_Object
VAR CONSTANT
    cMaxObjects1 : INT := 3;
END_VAR
VAR
    pSettings : POINTER TO ST_SettingMachinePart01;
END_VAR
VAR
    fbCylinder1_OneValve : FB_CylinderOneValveSpringRetX_2;
    fbCylinder1_TwoValve : FB_CylinderTwoValveRetX_3;
    fbMotor1_Motor : FB_Motor;
    fbMotor1_FI : FB_MotorInverterFITYPE;
    
    iCylinder1 : I_StandardCylinder;
    iMotor1 : I_StandardMotor;
	
	aObjects : ARRAY[0..cMaxObjects1] OF POINTER TO I_Object := [ADR(iCylinder1), ADR(iMotor1)];
	nLoop : INT;
END_VAR

METHOD INTERNAL Control
VAR_INPUT
END_VAR
{warning 'Add machine part cyclic control implementation'}

CASE pSettings^.nCylinderType OF
    0: 
        iCylinder1 := fbCylinder1_OneValve;
    1:
        iCylinder1 := fbCylinder1_TwoValve;
    ELSE
        iCylinder1 := fbCylinder1_OneValve;
END_CASE

CASE pSettings^.nMotorType OF
    0: 
        iMotor1 := fbMotor1_Motor;
    1:
        iMotor1 := fbMotor1_FI;
    ELSE
        iMotor1 := fbMotor1_Motor;
END_CASE


FOR nLoop := 0 TO cMaxObjects1 DO
    IF aObjects[nLoop] <> 0 THEN
		IF aObjects[nLoop]^ <> 0 THEN
			aObjects[nLoop]^.CycleTask();
		END_IF
	END_IF
END_FOR

SetError(nErrorID := 1);
END_METHOD

METHOD FB_init : BOOL
VAR_INPUT
	(* if TRUE, the retain variables are initialized (warm start / cold start)*)
	{attribute '''NORMAL__COMMENT' := ' if TRUE, the retain variables are initialized (warm start / cold start)'}
	bInitRetains	: BOOL;
	(* if TRUE, the instance afterwards gets moved into the copy code (online change)*)
	{attribute '''NORMAL__COMMENT' := ' if TRUE, the instance afterwards gets moved into the copy code (online change)'}
	bInCopyCode	: BOOL;
	(*Pointer to motor settings*)
	{attribute '''NORMAL__COMMENT' := 'Pointer to motor settings'}
	pSettings	: POINTER TO ST_SettingMachinePart01;
END_VAR
sName := 'FB_MachinePart01';
sVersion := '1.0.0.0';

THIS^.pSettings := pSettings;
END_METHOD

///Initialize FB, Override to do custom initialize, no need to call super
METHOD INTERNAL Init : HRESULT
{warning 'Add machine part init implementation'}

fbCylinder1_OneValve.Settings := ADR(pSettings^.stCylinderSettings);
fbCylinder1_TwoValve.Settings := ADR(pSettings^.stCylinderSettings);
fbMotor1_Motor.Settings  := ADR(pSettings^.stMotorSettings);
fbMotor1_FI.Settings  := ADR(pSettings^.stMotorSettings);

Init := GVL_HResultSuccess.cHR_SuccesDone;
END_METHOD

{attribute '''DOCU__COMMENT' := 'Reset error'}
(*Reset error*)
METHOD Reset
SUPER^.Reset();

{warning 'Add reset implementation'}
END_METHOD

END_FUNCTION_BLOCK

// ---- 991 - NTO Actuators/010 - Cylinders/CylinderCollection/FB_CylinderOneValveSpringRetX_2.TcPOU
{attribute 'c++_compatible'}
FUNCTION_BLOCK FB_CylinderOneValveSpringRetX_2 EXTENDS FB_Object IMPLEMENTS I_StandardCylinder
///In / outputs
VAR
    DO_bValve AT %Q* : BOOL;
    DI_bCylAtHome AT %I* : BOOL;
    DI_bCylAtOut AT %I* : BOOL;
END_VAR
VAR
    pSettings : POINTER TO ST_StandardCylinderSettings;
END_VAR

(*Cylinder at home position*)
PROPERTY AtHome : BOOL
GET
END_GET
END_PROPERTY

(*Cylinder at out position*)
PROPERTY AtOut : BOOL
GET
END_GET
END_PROPERTY

METHOD INTERNAL Control
VAR_INPUT
END_VAR
{warning 'Add valve cyclic control implementation'}
END_METHOD

(*Enable cylinder to change position*)
PROPERTY Enable : BOOL
GET
END_GET
SET
END_SET
END_PROPERTY

METHOD FB_init : BOOL
VAR_INPUT
	(* if TRUE, the retain variables are initialized (warm start / cold start)*)
	{attribute '''NORMAL__COMMENT' := ' if TRUE, the retain variables are initialized (warm start / cold start)'}
	bInitRetains	: BOOL;
	(* if TRUE, the instance afterwards gets moved into the copy code (online change)*)
	{attribute '''NORMAL__COMMENT' := ' if TRUE, the instance afterwards gets moved into the copy code (online change)'}
	bInCopyCode	: BOOL;
END_VAR
sName := 'FB_CylinderOneValveSpringRetX_2';
sVersion := '1.0.0.0';
END_METHOD

///Initialize FB, Override to do custom initialize, no need to call super
METHOD INTERNAL Init : HRESULT
Init := GVL_HResultSuccess.cHR_SuccesDone;
END_METHOD

METHOD MoveHome
END_METHOD

METHOD MoveOut
END_METHOD

{attribute '''DOCU__COMMENT' := 'Reset error, allways call super'}
(*Reset error, allways call super*)
METHOD Reset
SUPER^.Reset();

{warning 'Add reset implementation'}
END_METHOD

(*Pointer to settings, should be set at FB_init but can be modified with set accessor if needed*)
PROPERTY Settings : POINTER TO ST_StandardCylinderSettings
GET
Settings := pSettings;
END_GET
SET
pSettings := Settings;
END_SET
END_PROPERTY

END_FUNCTION_BLOCK

// ---- 991 - NTO Actuators/010 - Cylinders/CylinderCollection/FB_CylinderTwoValveRetX_3.TcPOU
{attribute 'c++_compatible'}
FUNCTION_BLOCK FB_CylinderTwoValveRetX_3 EXTENDS FB_Object IMPLEMENTS I_StandardCylinder
///In / outputs
VAR
    DO_bValve AT %Q* : BOOL;
    DI_bCylAtHome AT %I* : BOOL;
    DI_bCylAtOut AT %I* : BOOL;
END_VAR
VAR
    pSettings : POINTER TO ST_StandardCylinderSettings;
END_VAR

(*Cylinder at home position*)
PROPERTY AtHome : BOOL
GET
END_GET
END_PROPERTY

(*Cylinder at out position*)
PROPERTY AtOut : BOOL
GET
END_GET
END_PROPERTY

METHOD INTERNAL Control
VAR_INPUT
END_VAR
{warning 'Add valve cyclic control implementation'}
END_METHOD

(*Enable cylinder to change position*)
PROPERTY Enable : BOOL
GET
END_GET
SET
END_SET
END_PROPERTY

METHOD FB_init : BOOL
VAR_INPUT
	(* if TRUE, the retain variables are initialized (warm start / cold start)*)
	{attribute '''NORMAL__COMMENT' := ' if TRUE, the retain variables are initialized (warm start / cold start)'}
	bInitRetains	: BOOL;
	(* if TRUE, the instance afterwards gets moved into the copy code (online change)*)
	{attribute '''NORMAL__COMMENT' := ' if TRUE, the instance afterwards gets moved into the copy code (online change)'}
	bInCopyCode	: BOOL;
END_VAR
sName := 'FB_CylinderOneValveSpringRetX_2';
sVersion := '1.0.0.0';
END_METHOD

///Initialize FB, Override to do custom initialize, no need to call super
METHOD INTERNAL Init : HRESULT
Init := GVL_HResultSuccess.cHR_SuccesDone;
END_METHOD

METHOD MoveHome
END_METHOD

METHOD MoveOut
END_METHOD

{attribute '''DOCU__COMMENT' := 'Reset error, allways call super'}
(*Reset error, allways call super*)
METHOD Reset
SUPER^.Reset();

{warning 'Add reset implementation'}
END_METHOD

(*Pointer to settings, should be set at FB_init but can be modified with set accessor if needed*)
PROPERTY Settings : POINTER TO ST_StandardCylinderSettings
GET
Settings := pSettings;
END_GET
SET
pSettings := Settings;
END_SET
END_PROPERTY

END_FUNCTION_BLOCK

// ---- 991 - NTO Actuators/020 - Motors/MotorCollection/FB_Motor.TcPOU
{attribute 'c++_compatible'}
FUNCTION_BLOCK FB_Motor EXTENDS FB_Object IMPLEMENTS I_StandardMotor
///In / outputs
VAR
    DO_bCW AT %Q* : BOOL;
    DO_bCCW AT %Q* : BOOL;
    DI_bMotorOk AT %I* : BOOL := TRUE;
END_VAR
VAR
    bMoveCW : BOOL;
    bMoveCCW : BOOL;
    bEnable : BOOL;
    bLimitCW : BOOL;
    bLimitCCW : BOOL;
    nAcceleration : UINT;
    nDeceleration : UINT;
    nSpeed : UINT;
    pSettings : POINTER TO ST_StandardMotorSettings;
END_VAR

(*Accelaration in FI dependent type*)
PROPERTY Acc : UINT
GET
END_GET
SET
END_SET
END_PROPERTY

(*Move motor CCW*)
PROPERTY CCW : BOOL
GET
END_GET
SET
END_SET
END_PROPERTY

METHOD INTERNAL Control
VAR_INPUT
END_VAR
{warning 'Add motor cyclic control implementation'}
END_METHOD


(*Move motor CW*)
PROPERTY CW : BOOL
GET
END_GET
SET
END_SET
END_PROPERTY

(*Deceleration in FI dependent type*)
PROPERTY Dec : UINT
GET
END_GET
SET
END_SET
END_PROPERTY


(*Enable Motor*)
PROPERTY Enable : BOOL
GET
END_GET
SET
END_SET
END_PROPERTY

METHOD FB_init : BOOL
VAR_INPUT
	(* if TRUE, the retain variables are initialized (warm start / cold start)*)
	{attribute '''NORMAL__COMMENT' := ' if TRUE, the retain variables are initialized (warm start / cold start)'}
	bInitRetains	: BOOL;
	(* if TRUE, the instance afterwards gets moved into the copy code (online change)*)
	{attribute '''NORMAL__COMMENT' := ' if TRUE, the instance afterwards gets moved into the copy code (online change)'}
	bInCopyCode	: BOOL;
END_VAR
sName := 'FB_Motor';
sVersion := '1.0.0.0';
END_METHOD

///Initialize FB, Override to do custom initialize, no need to call super
METHOD INTERNAL Init : HRESULT
Init := GVL_HResultSuccess.cHR_SuccesDone;
END_METHOD

(*Limit counter-clockwise rotation*)
PROPERTY LimitCCW : BOOL
GET
END_GET
SET
END_SET
END_PROPERTY

(*Limit clockwise rotation*)
PROPERTY LimitCW : BOOL
GET
END_GET
SET
END_SET
END_PROPERTY

{attribute '''DOCU__COMMENT' := 'Reset error'}
(*Reset error*)
METHOD Reset
SUPER^.Reset();

{warning 'Add reset implementation'}
END_METHOD

(*Pointer to settings, should be set at FB_init but can be modified with set accessor if needed*)
PROPERTY Settings : POINTER TO ST_StandardMotorSettings
GET
Settings := pSettings;
END_GET
SET
pSettings := Settings;
END_SET
END_PROPERTY

(*Motor speed in 0.1 % *)
PROPERTY Speed : UINT
GET
END_GET
SET
END_SET
END_PROPERTY

END_FUNCTION_BLOCK

// ---- 991 - NTO Actuators/020 - Motors/MotorCollection/FB_MotorInverterFITYPE.TcPOU
{attribute 'c++_compatible'}
FUNCTION_BLOCK FB_MotorInverterFITYPE EXTENDS FB_Object IMPLEMENTS I_StandardMotor
///In / outputs
VAR
    DO_nControlWord AT %Q* : WORD;
    DO_nSpeed AT %Q* : WORD;
    DO_nRamp AT %Q* : WORD;
    DI_nStatusWord AT %I* : WORD;
    DI_nActSpeed AT %I* : WORD;
    DI_nCurrent AT %I* : WORD;
END_VAR
VAR
    bMoveCW : BOOL;
    bMoveCCW : BOOL;
    bEnable : BOOL;
    bLimitCW : BOOL;
    bLimitCCW : BOOL;
    nAcceleration : UINT;
    nDeceleration : UINT;
    nSpeed : UINT;
    pSettings : POINTER TO ST_StandardMotorSettings;
END_VAR

(*Accelaration in FI dependent type*)
PROPERTY Acc : UINT
GET
END_GET
SET
END_SET
END_PROPERTY

(*Move motor CCW*)
PROPERTY CCW : BOOL
GET
END_GET
SET
END_SET
END_PROPERTY

METHOD INTERNAL Control
VAR_INPUT
END_VAR
{warning 'Add motor cyclic control implementation'}
END_METHOD


(*Move motor CW*)
PROPERTY CW : BOOL
GET
END_GET
SET
END_SET
END_PROPERTY

(*Deceleration in FI dependent type*)
PROPERTY Dec : UINT
GET
END_GET
SET
END_SET
END_PROPERTY


(*Enable Motor*)
PROPERTY Enable : BOOL
GET
END_GET
SET
END_SET
END_PROPERTY

METHOD FB_init : BOOL
VAR_INPUT
	(* if TRUE, the retain variables are initialized (warm start / cold start)*)
	{attribute '''NORMAL__COMMENT' := ' if TRUE, the retain variables are initialized (warm start / cold start)'}
	bInitRetains	: BOOL;
	(* if TRUE, the instance afterwards gets moved into the copy code (online change)*)
	{attribute '''NORMAL__COMMENT' := ' if TRUE, the instance afterwards gets moved into the copy code (online change)'}
	bInCopyCode	: BOOL;
END_VAR
sName := 'FB_MotorInverterFITYPE';
sVersion := '1.0.0.0';
END_METHOD

///Initialize FB, Override to do custom initialize, no need to call super
METHOD INTERNAL Init : HRESULT
Init := GVL_HResultSuccess.cHR_SuccesDone;
END_METHOD

(*Limit counter-clockwise rotation*)
PROPERTY LimitCCW : BOOL
GET
END_GET
SET
END_SET
END_PROPERTY

(*Limit clockwise rotation*)
PROPERTY LimitCW : BOOL
GET
END_GET
SET
END_SET
END_PROPERTY

{attribute '''DOCU__COMMENT' := 'Reset error'}
(*Reset error*)
METHOD Reset
SUPER^.Reset();

{warning 'Add reset implementation'}
END_METHOD

(*Pointer to settings, should be set at FB_init but can be modified with set accessor if needed*)
PROPERTY Settings : POINTER TO ST_StandardMotorSettings
GET
Settings := pSettings;
END_GET
SET
pSettings := Settings;
END_SET
END_PROPERTY

(*Motor speed in 0.1 % *)
PROPERTY Speed : UINT
GET
END_GET
SET
END_SET
END_PROPERTY

END_FUNCTION_BLOCK

// ---- 020 - Machine Part 02/FB_MachinePart02.TcPOU
{attribute 'c++_compatible'}
FUNCTION_BLOCK FB_MachinePart02 EXTENDS FB_Object
VAR CONSTANT
    cMaxObjects1 : INT := 3;
END_VAR
VAR
    pSettings : POINTER TO ST_SettingMachinePart02;
END_VAR
VAR
    fbCylinder1_OneValve : FB_CylinderOneValveSpringRetX_2;
    fbCylinder1_TwoValve : FB_CylinderTwoValveRetX_3;
	iCylinder1 : I_StandardCylinder;
	
    fbCylinder2_OneValve : FB_CylinderOneValveSpringRetX_2;
    fbCylinder2_TwoValve : FB_CylinderTwoValveRetX_3;
	iCylinder2 : I_StandardCylinder;    
	
	aObjects : ARRAY[0..cMaxObjects1] OF POINTER TO I_Object := [ADR(iCylinder1), ADR(iCylinder2)];
	nLoop : INT;
END_VAR

METHOD INTERNAL Control
VAR_INPUT
END_VAR
{warning 'Add machine part cyclic control implementation'}

CASE pSettings^.nCylinder1Type OF
    0: 
        iCylinder1 := fbCylinder1_OneValve;
    1:
        iCylinder1 := fbCylinder1_TwoValve;
    ELSE
        iCylinder1 := fbCylinder1_OneValve;
END_CASE
CASE pSettings^.nCylinder2Type OF
    0: 
        iCylinder2 := fbCylinder2_OneValve;
    1:
        iCylinder2 := fbCylinder2_TwoValve;
    ELSE
        iCylinder2 := fbCylinder2_OneValve;
END_CASE




FOR nLoop := 0 TO cMaxObjects1 DO
    IF aObjects[nLoop] <> 0 THEN
		IF aObjects[nLoop]^ <> 0 THEN
			aObjects[nLoop]^.CycleTask();
		END_IF
	END_IF
END_FOR
END_METHOD

METHOD FB_init : BOOL
VAR_INPUT
	(* if TRUE, the retain variables are initialized (warm start / cold start)*)
	{attribute '''NORMAL__COMMENT' := ' if TRUE, the retain variables are initialized (warm start / cold start)'}
	bInitRetains	: BOOL;
	(* if TRUE, the instance afterwards gets moved into the copy code (online change)*)
	{attribute '''NORMAL__COMMENT' := ' if TRUE, the instance afterwards gets moved into the copy code (online change)'}
	bInCopyCode	: BOOL;
	(*Pointer to motor settings*)
	{attribute '''NORMAL__COMMENT' := 'Pointer to motor settings'}
	pSettings	: POINTER TO ST_SettingMachinePart02;
END_VAR
sName := 'FB_MachinePart02';
sVersion := '1.0.0.0';

THIS^.pSettings := pSettings;
END_METHOD

///Initialize FB, Override to do custom initialize, no need to call super
METHOD INTERNAL Init : HRESULT
{warning 'Add machine part init implementation'}
fbCylinder1_OneValve.Settings := ADR(pSettings^.stCylinder1Settings);
fbCylinder1_TwoValve.Settings := ADR(pSettings^.stCylinder1Settings);
                     
fbCylinder2_OneValve.Settings := ADR(pSettings^.stCylinder2Settings);
fbCylinder2_TwoValve.Settings := ADR(pSettings^.stCylinder2Settings);


Init := GVL_HResultSuccess.cHR_SuccesDone;
END_METHOD

{attribute '''DOCU__COMMENT' := 'Reset error'}
(*Reset error*)
METHOD Reset
SUPER^.Reset();

{warning 'Add reset implementation'}
END_METHOD

END_FUNCTION_BLOCK

// ---- 100 - Network/FB_CustomTcp.TcPOU
{attribute 'c++_compatible'}
FUNCTION_BLOCK FB_CustomTcp EXTENDS FB_SimpleTcpClient
VAR
	nRcvCnt : UDINT;
	sData : STRING(255);
END_VAR

METHOD FB_init : BOOL
VAR_INPUT
	bInitRetains : BOOL; // if TRUE, the retain variables are initialized (warm start / cold start)
	bInCopyCode : BOOL;  // if TRUE, the instance afterwards gets moved into the copy code (online change)
END_VAR
VAR
	ipSrv : ITComObjectServer;
END_VAR
sName := 'FB_CustomTcp';
sVersion := '1.0.0.0';
END_METHOD

END_FUNCTION_BLOCK

// ---- 100 - Network/SampleTcpClient.TcPOU
{attribute 'c++_compatible'}
FUNCTION_BLOCK SampleTcpClient EXTENDS FB_Object IMPLEMENTS ITcIoTcpProtocolRecv
VAR_INPUT
END_VAR
VAR_OUTPUT
END_VAR
VAR
	{attribute 'TcInitSymbol'}
	oid : OTCID;
	ipTcp : ITcIoTcpProtocol;
	socketID : UDINT;
	sendData : BOOL;
	dataToSend : U_Data := (sData := 'Sending from here');
	aLog : ARRAY[0..99] OF ST_Log;
	nLogEntry : INT := 0;
	aRcvData : ARRAY[0..99] OF U_Data;
	nRcvData : USINT;
	nPort : UINT := 9991;
	bConnect : BOOL;
	bIsConnected : BOOL;
	stIp : IPADDR := [41,1,168,192];
	uIP : U_IPAddr := (nIpAddr := 3232235817);
END_VAR

METHOD INTERNAL Control
VAR_INPUT
END_VAR
VAR
	nSendData : UDINT;
END_VAR
IF socketID <> 0 AND ipTcp <> 0 THEN
	bIsConnected := Tc3_Module.SUCCEEDED(ipTcp.IsConnected(socketId));
ELSE
	bIsConnected := FALSE;
END_IF
IF bConnect AND socketID = 0 THEN
	
	;//Open socket
	IF Tc3_Module.SUCCEEDED(ipTcp.AllocSocket(ipRecv := THIS^,socketId := socketID)) THEN
		
		IF Tc3_Module.FAILED(ipTcp.Connect(socketId := socketId, ipRemoteAddress := uIP.nIpAddr, tcpPort := nPort)) THEN
			ipTcp.FreeSocket(socketID);
			socketID := 0;
		END_IF 

	END_IF
	
ELSIF NOT(bConnect) AND socketID <> 0 THEN
	
	; //Close socket
	IF Tc3_Module.SUCCEEDED(ipTcp.IsConnected(socketId)) THEN
		ipTcp.Close(socketId);
		ipTcp.CheckReceived();
	END_IF
	ipTcp.FreeSocket(socketId);
	socketId := 0;
	
ELSIF bConnect AND socketID <> 0 THEN

	;//Check if send data 
	IF bIsConnected AND sendData THEN
		nSendData := 0;
		ipTcp.SendData(socketId := socketID, nData := SIZEOF(dataToSend), pData := ADR(dataToSend), nSendData := nSendData);
		sendData := FALSE;
	END_IF
	
END_IF

ipTcp.CheckReceived();
END_METHOD

METHOD FB_exit : BOOL
VAR_INPUT
	bInCopyCode : BOOL; // if TRUE, the exit method is called for exiting an instance that is copied afterwards (online change).
END_VAR
IF ipTcp <> 0 THEN
	IF socketID <> 0 THEN
		IF Tc3_Module.SUCCEEDED(ipTcp.IsConnected(socketId)) THEN
			ipTcp.Close(socketId);
			ipTcp.CheckReceived();
		END_IF
		ipTcp.FreeSocket(socketId);
		socketId := 0;
	ELSE
		FB_exit := TRUE;
	END_IF
ELSE
	FB_exit := FALSE;	
END_IF
END_METHOD

METHOD FB_init : BOOL
VAR_INPUT
	bInitRetains : BOOL; // if TRUE, the retain variables are initialized (warm start / cold start)
	bInCopyCode : BOOL;  // if TRUE, the instance afterwards gets moved into the copy code (online change)
END_VAR
VAR
	ipSrv : ITComObjectServer;
END_VAR
sName := 'SampleTcpClient';
sVersion := '1.0.0.0';

IF Tc3_Module.FW_ObjMgr_GetObjectServer(oidApp := _AppInfo.ObjId, pipSrv := ADR(ipSrv)) = Tc3_Module.S_OK THEN
	
	IF ipSrv.TcQueryObjectInterface(oid := oid, iid := IID_ITcIoTcpProtocol, ADR(ipTcp)) = Tc3_Module.S_OK THEN
		FB_init := TRUE;
	ELSE
		FB_init := FALSE;
	END_IF
	ipSrv.TcRelease();
	ipSrv := 0;
ELSE
	FB_init := FALSE;
END_IF
END_METHOD

{attribute 'c++_compatible'}
{attribute 'signature_flag' := '33554688'}
{attribute 'pack_mode' := '4'}
{attribute 'show'}
{attribute 'minimal_input_size' := '4'}
{attribute 'checksuperglobal'}
METHOD ReceiveData : HRESULT
VAR_INPUT
	socketId	: UDINT;
	nData	: UDINT;
	pData	: PVOID;
END_VAR
Tc2_System.MEMCPY(ADR(aRcvData[nRcvData]),pData,MIN(255,nData));
nRcvData := nRcvData + 1;


IF nRcvData > 99 THEN
	nRcvData := 0;
END_IF
END_METHOD

{attribute 'c++_compatible'}
{attribute 'signature_flag' := '33554688'}
{attribute 'pack_mode' := '4'}
{attribute 'show'}
{attribute 'minimal_input_size' := '4'}
{attribute 'checksuperglobal'}
METHOD ReceiveEvent : HRESULT
VAR_INPUT
	socketId	: UDINT;
	tcpEvent	: TCPIP_EVENT;
END_VAR
aLog[nLogEntry].eTcpEvent := tcpEvent;
aLog[nLogEntry].nSocketID := socketId;
nLogEntry := nLogEntry + 1;
IF nLogEntry > 99 THEN
	nLogEntry := 0;
END_IF

IF tcpEvent = TCPIP_EVENT.TCPIP_EVENT_CONN_CLOSED THEN
	bConnect := FALSE;
END_IF
END_METHOD

{attribute 'c++_compatible'}
{attribute 'signature_flag' := '33554688'}
{attribute 'pack_mode' := '4'}
{attribute 'show'}
{attribute 'minimal_input_size' := '4'}
{attribute 'checksuperglobal'}
METHOD TcAddRef : UDINT
END_METHOD

{attribute 'c++_compatible'}
{attribute 'signature_flag' := '33554688'}
{attribute 'pack_mode' := '4'}
{attribute 'show'}
{attribute 'minimal_input_size' := '4'}
{attribute 'checksuperglobal'}
METHOD TcQueryInterface : HRESULT
VAR_INPUT
	iid	: REFERENCE TO IID;
	pipItf	: POINTER TO PVOID;
END_VAR
END_METHOD

{attribute 'c++_compatible'}
{attribute 'signature_flag' := '33554688'}
{attribute 'pack_mode' := '4'}
{attribute 'show'}
{attribute 'minimal_input_size' := '4'}
{attribute 'checksuperglobal'}
METHOD TcRelease : UDINT
END_METHOD

END_FUNCTION_BLOCK

// ---- 100 - Network/SampleTcpServer.TcPOU
{attribute 'c++_compatible'}
FUNCTION_BLOCK SampleTcpServer EXTENDS FB_Object IMPLEMENTS ITcIoTcpProtocolRecv
VAR_INPUT
END_VAR
VAR_OUTPUT
END_VAR
VAR
	{attribute 'TcInitSymbol'}
	oid : OTCID;
	ipTcp : ITcIoTcpProtocol;
	socketID : UDINT;
	sendData : BOOL;
	dataToSend : U_Data := (sData := 'Sending from here');
	aLog : ARRAY[0..99] OF ST_Log;
	nLogEntry : INT := 0;
	aRcvData : ARRAY[0..99] OF U_Data;
	nRcvData : USINT;
	nPort : UINT := 9992;
	bConnect : BOOL;
	bIsConnected : BOOL;
	uRemoteIP : U_IPAddr;
	nConnectedSocket : UDINT;
END_VAR
VAR
	nSendData : UDINT;
END_VAR
VAR
	nSendData1 : UDINT;
	nSendData2 : UDINT;
END_VAR

METHOD INTERNAL Control
VAR_INPUT
END_VAR
IF socketID <> 0 AND ipTcp <> 0 THEN
	bIsConnected := Tc3_Module.SUCCEEDED(ipTcp.IsConnected(socketId));
ELSE
	bIsConnected := FALSE;
END_IF
IF bConnect AND socketID = 0 THEN
	;//Open socket
	IF Tc3_Module.SUCCEEDED(ipTcp.AllocSocket(ipRecv := THIS^,socketId := socketID)) THEN		
		
		IF Tc3_Module.FAILED(ipTcp.Listen(socketId := socketId, tcpPort := nPort)) THEN
			ipTcp.FreeSocket(socketID);
			socketID := 0;
		END_IF 

	END_IF
	
ELSIF NOT(bConnect) AND socketID <> 0 THEN
	
	; //Close socket
	IF Tc3_Module.SUCCEEDED(ipTcp.IsConnected(socketId)) THEN
		ipTcp.Close(socketId);
		ipTcp.CheckReceived();
	END_IF
	ipTcp.FreeSocket(socketId);
	socketId := 0;
	
ELSIF bConnect AND socketID <> 0 THEN

	;//Check if send data 
	IF bIsConnected AND sendData THEN
		nSendData := 0;
		ipTcp.SendData(socketId := nConnectedSocket, nData := SIZEOF(dataToSend), pData := ADR(dataToSend), nSendData := nSendData);
		sendData := FALSE;
	END_IF
	
END_IF

ipTcp.CheckReceived();
END_METHOD

METHOD FB_exit : BOOL
VAR_INPUT
	bInCopyCode : BOOL; // if TRUE, the exit method is called for exiting an instance that is copied afterwards (online change).
END_VAR
IF ipTcp <> 0 THEN
	IF socketID <> 0 THEN
		IF Tc3_Module.SUCCEEDED(ipTcp.IsConnected(socketId)) THEN
			ipTcp.Close(socketId);
			ipTcp.CheckReceived();
		END_IF
		ipTcp.FreeSocket(socketId);
		socketId := 0;
	ELSE
		FB_exit := TRUE;
	END_IF
ELSE
	FB_exit := FALSE;	
END_IF
END_METHOD

METHOD FB_init : BOOL
VAR_INPUT
	bInitRetains : BOOL; // if TRUE, the retain variables are initialized (warm start / cold start)
	bInCopyCode : BOOL;  // if TRUE, the instance afterwards gets moved into the copy code (online change)
END_VAR
VAR
	ipSrv : ITComObjectServer;
END_VAR
sName := 'SampleTcpServer';
sVersion := '1.0.0.0';

IF Tc3_Module.FW_ObjMgr_GetObjectServer(oidApp := _AppInfo.ObjId, pipSrv := ADR(ipSrv)) = Tc3_Module.S_OK THEN
	
	IF ipSrv.TcQueryObjectInterface(oid := oid, iid := IID_ITcIoTcpProtocol, ADR(ipTcp)) = Tc3_Module.S_OK THEN
		FB_init := TRUE;
	ELSE
		FB_init := FALSE;
	END_IF
	ipSrv.TcRelease();
	ipSrv := 0;
ELSE
	FB_init := FALSE;
END_IF
END_METHOD

{attribute 'c++_compatible'}
{attribute 'signature_flag' := '33554688'}
{attribute 'pack_mode' := '4'}
{attribute 'show'}
{attribute 'minimal_input_size' := '4'}
{attribute 'checksuperglobal'}
METHOD ReceiveData : HRESULT
VAR_INPUT
	socketId	: UDINT;
	nData	: UDINT;
	pData	: PVOID;
END_VAR
VAR
	uData : U_Data := (sData := 'Did you send to me?$n$r'); 
END_VAR
Tc2_System.MEMCPY(ADR(aRcvData[nRcvData]),pData,MIN(255,nData));

ipTcp.SendData(socketId := socketId, nData := SIZEOF(uData), pData := ADR(uData), nSendData := nSendData1);
ipTcp.SendData(socketId := socketId, nData := SIZEOF(aRcvData[nRcvData]), pData := ADR(aRcvData[nRcvData]), nSendData := nSendData2);

nRcvData := nRcvData + 1;
IF nRcvData > 99 THEN
	nRcvData := 0;
END_IF

ipTcp.GetRemoteIpAddr(socketId := socketId, remoteIpAddr := uRemoteIP.nIpAddr);
END_METHOD

{attribute 'c++_compatible'}
{attribute 'signature_flag' := '33554688'}
{attribute 'pack_mode' := '4'}
{attribute 'show'}
{attribute 'minimal_input_size' := '4'}
{attribute 'checksuperglobal'}
METHOD ReceiveEvent : HRESULT
VAR_INPUT
	socketId	: UDINT;
	tcpEvent	: TCPIP_EVENT;
END_VAR
aLog[nLogEntry].eTcpEvent := tcpEvent;
aLog[nLogEntry].nSocketID := socketId;
nLogEntry := nLogEntry + 1;
IF nLogEntry > 99 THEN
	nLogEntry := 0;
END_IF
CASE tcpEvent OF
	TCPIP_EVENT.TCPIP_EVENT_CONN_INCOMING :
		ipTcp.Accept(socketId);
		nConnectedSocket := socketID;
	TCPIP_EVENT.TCPIP_EVENT_CONN_CLOSED :
		
END_CASE
END_METHOD

{attribute 'c++_compatible'}
{attribute 'signature_flag' := '33554688'}
{attribute 'pack_mode' := '4'}
{attribute 'show'}
{attribute 'minimal_input_size' := '4'}
{attribute 'checksuperglobal'}
METHOD TcAddRef : UDINT
END_METHOD

{attribute 'c++_compatible'}
{attribute 'signature_flag' := '33554688'}
{attribute 'pack_mode' := '4'}
{attribute 'show'}
{attribute 'minimal_input_size' := '4'}
{attribute 'checksuperglobal'}
METHOD TcQueryInterface : HRESULT
VAR_INPUT
	iid	: REFERENCE TO IID;
	pipItf	: POINTER TO PVOID;
END_VAR
END_METHOD

{attribute 'c++_compatible'}
{attribute 'signature_flag' := '33554688'}
{attribute 'pack_mode' := '4'}
{attribute 'show'}
{attribute 'minimal_input_size' := '4'}
{attribute 'checksuperglobal'}
METHOD TcRelease : UDINT
END_METHOD

END_FUNCTION_BLOCK

// ---- 100 - Network/SampleUdpEchoServer.TcPOU
{attribute 'c++_compatible'}
FUNCTION_BLOCK SampleUdpEchoServer IMPLEMENTS ITcIoUdpProtocolRecv
VAR_INPUT
END_VAR
VAR_OUTPUT
END_VAR
VAR	
	{attribute 'TcInitSymbol'}
	oid : OTCID;
	ipUdp : ITcIoUdpProtocol;
	udpPort : UINT := 10000;
	nRecievedPackets : UINT;
END_VAR

IF ipUdp <> 0 THEN
	ipUdp.CheckReceived();
END_IF

METHOD FB_exit : BOOL
VAR_INPUT
	bInCopyCode : BOOL; // if TRUE, the exit method is called for exiting an instance that is copied afterwards (online change).
END_VAR
IF ipUdp <> 0 THEN
	ipUdp.UnregisterReceiver(udpPort);
	ipUdp.TcRelease();
	ipUdp := 0;
	FB_exit := TRUE;
ELSE
	FB_exit := FALSE;
END_IF
END_METHOD

METHOD FB_init : BOOL
VAR_INPUT
	bInitRetains : BOOL; // if TRUE, the retain variables are initialized (warm start / cold start)
	bInCopyCode : BOOL;  // if TRUE, the instance afterwards gets moved into the copy code (online change)
END_VAR
VAR
	ipSrv : ITComObjectServer;
END_VAR
IF Tc3_Module.FW_ObjMgr_GetObjectServer(oidApp := _AppInfo.ObjId, pipSrv := ADR(ipSrv)) = Tc3_Module.S_OK THEN
	
	IF ipSrv.TcQueryObjectInterface(oid := oid, iid := IID_ITcIoUdpProtocol, ADR(ipUdp)) = Tc3_Module.S_OK THEN
		
		IF ipUdp.RegisterReceiver(udpPort := udpPort, ipRecv := THIS^) = 0 THEN
			FB_init := FALSE;
		ELSE
			FB_init := FALSE;
			ipUdp.TcRelease();
			ipUdp := 0;
		END_IF
	ELSE
		FB_init := FALSE;
	END_IF
	ipSrv.TcRelease();
	ipSrv := 0;
ELSE
	FB_init := FALSE;
END_IF
END_METHOD

{attribute 'c++_compatible'}
{attribute 'signature_flag' := '33554688'}
{attribute 'pack_mode' := '4'}
{attribute 'show'}
{attribute 'minimal_input_size' := '4'}
{attribute 'checksuperglobal'}
METHOD ReceiveData : HRESULT
VAR_INPUT
	ipAddr	: UDINT;
	udpDestPort	: UINT;
	udpSrcPort	: UINT;
	nData	: UDINT;
	pData	: PVOID;
	pVlan	: POINTER TO ETYPE_VLAN_HEADER := 0;
END_VAR
nRecievedPackets := nRecievedPackets + 1;
IF ipUdp <> 0 THEN
	ipUdp.SendData(ipDestAddr := ipAddr,
					udpDestPort := udpSrcPort,
					udpSrcPort := udpDestPort,
					nData := nData,
					pData := pData,
					bCalcUdpCheckSum := TRUE,
					pVlan  := 0);	
END_IF
END_METHOD

{attribute 'c++_compatible'}
{attribute 'signature_flag' := '33554688'}
{attribute 'pack_mode' := '4'}
{attribute 'show'}
{attribute 'minimal_input_size' := '4'}
{attribute 'checksuperglobal'}
METHOD TcAddRef : UDINT
END_METHOD

{attribute 'c++_compatible'}
{attribute 'signature_flag' := '33554688'}
{attribute 'pack_mode' := '4'}
{attribute 'show'}
{attribute 'minimal_input_size' := '4'}
{attribute 'checksuperglobal'}
METHOD TcQueryInterface : HRESULT
VAR_INPUT
	iid	: REFERENCE TO IID;
	pipItf	: POINTER TO PVOID;
END_VAR
END_METHOD

{attribute 'c++_compatible'}
{attribute 'signature_flag' := '33554688'}
{attribute 'pack_mode' := '4'}
{attribute 'show'}
{attribute 'minimal_input_size' := '4'}
{attribute 'checksuperglobal'}
METHOD TcRelease : UDINT
END_METHOD

END_FUNCTION_BLOCK

// ---- 990 - NTO Standard/HResult/F_Busy.TcPOU
///Checks if the returned HRESULT is success and busy
FUNCTION F_Busy : BOOL
VAR_INPUT
    hr : HRESULT;
END_VAR
VAR
END_VAR

F_Busy := (hr = GVL_HResultSuccess.cHR_SuccesBusy);

END_FUNCTION

// ---- 990 - NTO Standard/HResult/F_Code.TcPOU
///Get the Code from the HRESULT
FUNCTION F_Code : UINT
VAR_INPUT
    hr : HRESULT;
END_VAR
VAR
END_VAR

F_Code := UDINT_TO_UINT(DINT_TO_UDINT(hr) AND 16#0000FFFF);

END_FUNCTION

// ---- 990 - NTO Standard/HResult/F_Fail.TcPOU
///Checks if the HRESULT is error
FUNCTION F_Fail : BOOL
VAR_INPUT
    hr : HRESULT;
END_VAR
VAR
END_VAR

F_Fail := (hr < 0);

END_FUNCTION

// ---- 990 - NTO Standard/HResult/F_Success.TcPOU
///Checks if the returned HRESULT is success
FUNCTION F_Success : BOOL
VAR_INPUT
    hr : HRESULT;
END_VAR
VAR
END_VAR

F_Success := (hr >= 0);

END_FUNCTION

// ---- 000 - General/visMain.TcVIS
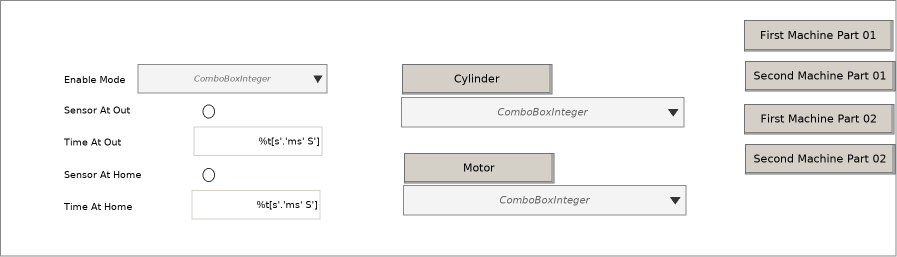
VISUALIZATION visMain  // 897x257
VAR_IN_OUT
	
END_VAR
VAR
	nSel : INT := 0;
END_VAR
    Frame (21,20 713x235)
        shows visSettingMachPart1(refSetting := MAIN.fbMach01_1.pSettings^)
        shows visSettingMachPart1(refSetting := MAIN.fbMach01_2.pSettings^)
        shows visSettingMachPart2(refSetting := MAIN.fbMach02_1.pSettings^)
        shows visSettingMachPart2(refSetting := MAIN.fbMach02_2.pSettings^)
    Button (744,20 149x31), "First Machine Part 01", colour toggle: nSel = 0
        OnMouseClick: FrameSelectionChange Selection=SelectedFrame=4000cae3-cddb-40df-befc-2ce2e2612873, GlobSel=AssignType=Directly, SelType=Locally
        OnMouseClick: execute { nSel := 0; }
    Button (745,61 150x30), "Second Machine Part 01", colour toggle: nSel = 1
        OnMouseClick: FrameSelectionChange Selection=SelectedFrame=4000cae3-cddb-40df-befc-2ce2e2612873, Selection=1, GlobSel=AssignType=Directly, SelType=Locally
        OnMouseClick: execute { nSel := 1; }
    Button (744,104 150x30), "First Machine Part 02", colour toggle: nSel = 2
        OnMouseClick: FrameSelectionChange Selection=SelectedFrame=4000cae3-cddb-40df-befc-2ce2e2612873, Selection=2, GlobSel=AssignType=Directly, SelType=Locally
        OnMouseClick: execute { nSel := 2; }
    Button (745,144 150x30), "Second Machine Part 02", colour toggle: nSel = 3
        OnMouseClick: FrameSelectionChange Selection=SelectedFrame=4000cae3-cddb-40df-befc-2ce2e2612873, Selection=3, GlobSel=AssignType=Directly, SelType=Locally
        OnMouseClick: execute { nSel := 3; }
END_VISUALIZATION

// ---- 010 - Machine Part 01/visSettingMachPart1.TcVIS
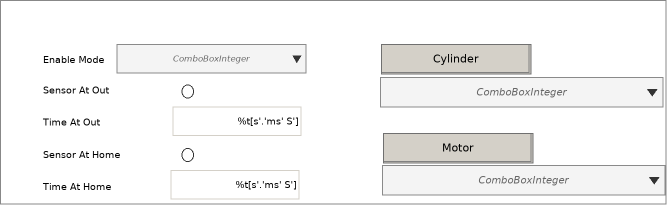
VISUALIZATION visSettingMachPart1  // 667x205
VAR_INPUT
	refSetting : REFERENCE TO ST_SettingMachinePart01;
END_VAR
VAR
	nSel : INT;
END_VAR
    Frame (31,30 277x173)
        shows visStandardCylinderSettings(refSetting := refSetting.stCylinderSettings)
        shows visStandardMotorSettings(refSetting := refSetting.stMotorSettings)
    Button (381,44 150x30), "Cylinder", colour toggle: nSel = 0
        OnMouseClick: FrameSelectionChange Selection=SelectedFrame=f571b872-985a-4510-9730-37c9a5269c7f, GlobSel=AssignType=Directly, SelType=Locally
        OnMouseClick: execute { nSel := 0; }
    Button (383,133 150x30), "Motor", colour toggle: nSel = 1
        OnMouseClick: FrameSelectionChange Selection=SelectedFrame=f571b872-985a-4510-9730-37c9a5269c7f, Selection=1, GlobSel=AssignType=Directly, SelType=Locally
        OnMouseClick: execute { nSel := 1; }
    ComboBoxInteger (380,77 283x30), variable: refSetting.nCylinderType, text list: 'txtCylinderTypes'
    ComboBoxInteger (382,165 283x30), variable: refSetting.nMotorType, text list: 'txtMotorTypes'
END_VISUALIZATION

// ---- 020 - Machine Part 02/visSettingMachPart2.TcVIS
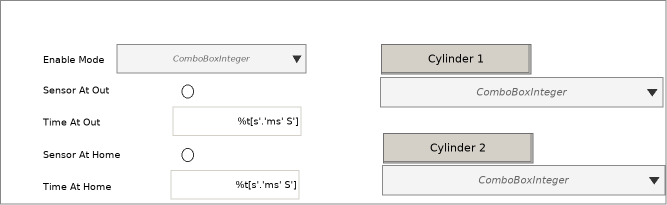
VISUALIZATION visSettingMachPart2  // 667x205
VAR_INPUT
	refSetting : REFERENCE TO ST_SettingMachinePart02;
END_VAR
VAR
	nSel : INT;
END_VAR
    Frame (31,30 277x173)
        shows visStandardCylinderSettings(refSetting := refSetting.stCylinder1Settings)
        shows visStandardCylinderSettings(refSetting := refSetting.stCylinder2Settings)
    Button (381,44 150x30), "Cylinder 1", colour toggle: nSel = 0
        OnMouseClick: FrameSelectionChange Selection=SelectedFrame=f571b872-985a-4510-9730-37c9a5269c7f, GlobSel=AssignType=Directly, SelType=Locally
        OnMouseClick: execute { nSel := 0; }
    Button (383,133 150x30), "Cylinder 2", colour toggle: nSel = 1
        OnMouseClick: FrameSelectionChange Selection=SelectedFrame=f571b872-985a-4510-9730-37c9a5269c7f, Selection=1, GlobSel=AssignType=Directly, SelType=Locally
        OnMouseClick: execute { nSel := 1; }
    ComboBoxInteger (380,77 283x30), variable: refSetting.nCylinder1Type, text list: 'txtCylinderTypes'
    ComboBoxInteger (382,165 283x30), variable: refSetting.nCylinder2Type, text list: 'txtCylinderTypes'
END_VISUALIZATION

// ---- 991 - NTO Actuators/010 - Cylinders/CylinderCollection/txtCylinderTypes.TcTLO
TEXTLIST txtCylinderTypes
  0 = 'One Valve Spring Ret X2'
  1 = 'Two Valve Ret X3'
   = ''
END_TEXTLIST

// ---- 991 - NTO Actuators/010 - Cylinders/txtLstCylinderEnableMode.TcTLO
TEXTLIST txtLstCylinderEnableMode
  0 = 'Off'
  1 = 'To Home'
  2 = 'To Out'
  3 = 'No Change Allowed'
   = ''
END_TEXTLIST

// ---- 991 - NTO Actuators/010 - Cylinders/visStandardCylinderSettings.TcVIS
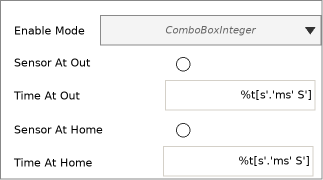
VISUALIZATION visStandardCylinderSettings  // 323x180
VAR_INPUT
	refSetting : REFERENCE TO ST_StandardCylinderSettings;
END_VAR
VAR CONSTANT
	cMinTime : DINT := 0;
	cMaxTime : DINT := T#100S;
	sDialog1 : STRING := 'Time at out';
	sDialog2 : STRING := 'Time at home';
END_VAR
    Label (11,48 150x30), "Sensor At Out"
    Label (11,81 150x30), "Time At Out"
    Label (11,148 150x30), "Time At Home"
    Label (11,115 150x30), "Sensor At Home"
    RadioButton (174,49 132x30), variable: refSetting.bSensorAtOut
        Areas[0]: Text=Off
        Areas[1]: Text=On
    Label (11,16 150x30), "Enable Mode"
    ComboBoxInteger (100,15 221x30), variable: refSetting.eEnableMode, text list: 'txtLstCylinderEnableMode'
    RadioButton (174,115 132x30), variable: refSetting.bSensorAtHome
        Areas[0]: Text=Off
        Areas[1]: Text=On
    Textfield (163,146 150x30), "%t[s'.'ms' S']", text variable: refSetting.tTimeToOrAtHome
        OnMouseClick: write the text variable via Default, min cMinTime, max cMaxTime, title sDialog2
    Textfield (165,80 150x30), "%t[s'.'ms' S']", text variable: refSetting.tTimeToOrAtOut
        OnMouseClick: write the text variable via Default, min cMinTime, max cMaxTime, title sDialog1
END_VISUALIZATION

// ---- 991 - NTO Actuators/020 - Motors/MotorCollection/txtMotorTypes.TcTLO
TEXTLIST txtMotorTypes
  0 = 'Contactor'
  1 = 'FI'
   = ''
END_TEXTLIST

// ---- 991 - NTO Actuators/020 - Motors/txtLstMotorEnableMode.TcTLO
TEXTLIST txtLstMotorEnableMode
  0 = 'Off'
  1 = 'Both Dir'
  2 = 'Only CW'
  3 = 'Only CCW'
   = ''
END_TEXTLIST

// ---- 991 - NTO Actuators/020 - Motors/visStandardMotorSettings.TcVIS
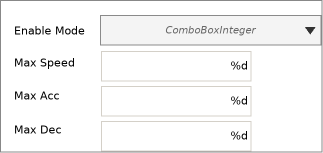
VISUALIZATION visStandardMotorSettings  // 323x153
VAR_INPUT
	refSetting : REFERENCE TO ST_StandardMotorSettings;
END_VAR
VAR CONSTANT
	cMinSpeed : UINT := 0;
	cMaxSpeed : UINT := 1000;
	cMinAcc : UINT := 1;
	cMaxAcc : UINT := 10000;
	cMinDec : UINT := 1;
	cMaxDec : UINT := 10000;
	cDialog1 : STRING := 'Max Speed in 0.1%';
	cDialog2 : STRING := 'Max Acc';
	cDialog3 : STRING := 'Max Dec';
END_VAR
    Label (11,48 150x30), "Max Speed"
    Label (11,81 150x30), "Max Acc"
    Label (11,115 150x30), "Max Dec"
    Label (11,16 150x30), "Enable Mode"
    ComboBoxInteger (100,15 221x30), variable: refSetting.eEnableMode, text list: 'txtLstMotorEnableMode'
    Textfield (101,51 150x30), "%d", text variable: refSetting.nMaxSpeed
        OnMouseClick: write the text variable via Default, min cMinSpeed, max cMaxSpeed, title cDialog1
    Textfield (101,86 150x30), "%d", text variable: refSetting.nMaxAcc
        OnMouseClick: write the text variable via Default, min cMinAcc, max cMaxAcc, title cDialog2
    Textfield (101,121 150x30), "%d", text variable: refSetting.nMaxDec
        OnMouseClick: write the text variable via Default, min cMinDec, max cMaxDec, title cDialog3
END_VISUALIZATION

// ---- GlobalTextList.TcGTLO
TEXTLIST GlobalTextList
  4 = ''
  29 = '%d'
  5 = '%d ms'
  25 = '%s'
  13 = '%t'
  11 = '%t ms'
  21 = "%t['ss'S'ms' ms']"
  20 = "%t[hh'h'mm'm'ss'S'ms' ms']"
  12 = '%t[HH:MM:SS] ms'
  16 = '%t[mm:ss:ms]'
  15 = '%t[ms]'
  24 = "%t[s'.'ms' S']"
  19 = "%t[ss' S 'ms' ms']"
  23 = "%t[ss'.'ms' S']"
  22 = "%t[ss'S'ms' ms']"
  18 = "%t[ss'S'ms'ms']"
  17 = '%t[ssms] ms'
  14 = '%t[]'
  7 = 'button 1'
  8 = 'button 2'
  30 = 'Cylinder'
  34 = 'Cylinder 1'
  35 = 'Cylinder 2'
  6 = 'Enable Mode'
  36 = 'First Machine Part 01'
  38 = 'First Machine Part 02'
  33 = 'Machine Part 01'
  32 = 'Machine Part 1'
  27 = 'Max Acc'
  28 = 'Max Dec'
  26 = 'Max Speed'
  31 = 'Motor'
  10 = 'Off'
  9 = 'On'
  37 = 'Second Machine Part 01'
  39 = 'Second Machine Part 02'
  1 = 'Sensor At Home'
  0 = 'Sensor At Out'
  3 = 'Time At Home'
  2 = 'Time At Out'
END_TEXTLIST
